// TIA Portal V16 export
// export: Created 2025-08-30T12:59:14.6807846Z, ExportSetting WithDefaults, DisplayName Totally Integrated Automation Portal, DisplayVersion V16, DisplayName TIA Portal Version Control Interface, DisplayVersion V16, DisplayName TIA Portal Openness, DisplayVersion V16, DisplayName STEP 7 Professional, DisplayVersion V16, DisplayName STEP 7 Safety, DisplayVersion V16, DisplayName WinCC Advanced, DisplayVersion V16
DATA_BLOCK "DB1"   // DB93
VERSION : 0.1
// stored: AutoNumber true, IsOnlyStoredInLoadMemory false, IsWriteProtectedInAS false
   VAR RETAIN
      DBB0 : DWord;
      DBB15 : DWord;
      DBB14 : DWord;
      DBB13 : DWord;
      DBB12 : DWord;
      DBB11 : DWord;
      DBB10 : DWord;
      DBB9 : DWord;
      DBB8 : DWord;
      DBB7 : DWord;
      DBB6 : DWord;
      DBB5 : DWord;
      DBB4 : DWord;
      DBB3 : DWord;
      DBB2 : DWord;
      DBB1 : DWord;
      DBD4 : DWord;
      DBD0 : DWord;
      "DBX4.0" : Bool;
   END_VAR
BEGIN
END_DATA_BLOCK
